FUNCTION_BLOCK PUBLIC FB_FIND_FILES
VAR_IN_OUT
	Filenames : ARRAY[*] OF STRING;
END_VAR
VAR_INPUT
	Filter : STRING;
	Execute : BOOL;
	Abort : BOOL;
END_VAR
VAR_OUTPUT
	Busy : BOOL;
	Done : BOOL;
	Error : BOOL;
END_VAR
VAR
	State : INT;
	i : DINT;
	FindFile : FB_EnumFindFileEntry;
END_VAR

CASE State OF 
	0: 
		Busy := FALSE;
		IF Execute THEN
			Done := FALSE;
			Error := FALSE;
			Busy := TRUE;
			Execute := FALSE;
			FindFile.eCmd := eEnumCmd_First;
			FindFile.sPathName := Filter;
			
			FOR i := LOWER_BOUND(Filenames, 1) TO UPPER_BOUND(Filenames, 1) DO
				Filenames[i] := '';
			END_FOR;
			
			i := LOWER_BOUND(Filenames, 1);
			State := 10;
		END_IF;
		
	10:
		IF Abort THEN
            Abort      := FALSE;
            FindFile.eCmd := eEnumCmd_Abort;
        END_IF
        FindFile(bExecute := FALSE);
        FindFile(bExecute := TRUE);
        State := 20;
		
	20:
		FindFile(bExecute := FALSE);
        IF NOT FindFile.bBusy THEN
            IF NOT FindFile.bError THEN
                IF NOT FindFile.bEOE AND i <= UPPER_BOUND(Filenames, 1) THEN
					Filenames[i] := FindFile.stFindFile.sFileName;
					i := i + 1;
					FindFile.eCmd := eEnumCmd_Next;
					State := 10;
                ELSE
					Done := TRUE;
                    State := 0;
                END_IF
            ELSE
                Error := TRUE;
                State     := 0;
            END_IF
        END_IF
END_CASE;

END_FUNCTION_BLOCK

(* stored: Version 1.1.0.1, ProductVersion 3.1.4024.12
   POU FB_FIND_FILES: Id {1e92509d-c6a4-4950-af30-a75beb75dab4}, SpecialFunc None *)
